{attribute 'qualified_only'}
{attribute 'strict'}
TYPE L_Stopper :
(
    ST1L0 := 1, // ST1
    ST1L1 := 2, // TXI PPS Stopper in
    MR1L0_L0 := 3, // MR1L0 Pitch state delivery to L0 line
    MR1L0_TXI := 4, //MR1L0 Pitch state delivery to TXI line
    MR1L1_IN:= 5, //  TXI Offset Mirror horizontal state
    MR1L1_OUT:= 6, // TXI Offset Mirror horizontal state
    ST1L2 := 7, // ST1L2 XPP Stopper
    XPP_SB23_MONO:=8, // Indicates that XPP SB2/3 is in MONO Line
    XPP_SB23_PINK:=9, //Indicates that XPP SB2/3 is in PINK Line
    XPP_SB6_MONO:=10, // Indicates that XPP SB6is in MONO Line
    XPP_SB6_PINK:=11, //Indicates that XPP SB6 is in PINK Line
    ST2L0 := 12, // ST2L0 XRT Stopper
    DEFAULT := PMPS_GVL.MAX_VETO_DEVICES // DO NOT USE FOR ANYTHING
);
END_TYPE

(* stored: Version 1.1.0.1
   DUT L_Stopper: Id {4f388ccc-0324-4da3-97c4-cae9c87c18e4} *)
